INTERFACE I_JsonDeserializerChangedEvent EXTENDS I_Event

PROPERTY PUBLIC Target : I_JsonDeserializer
GET
END_GET
END_PROPERTY

END_INTERFACE

(* stored: Version 1.1.0.1, ProductVersion 3.1.4024.12
   Itf I_JsonDeserializerChangedEvent: Id {40baa505-43af-4f39-bb65-a6df1e3a04e2}
   Property Target: Id {c8ae607c-6e4e-4a76-b1e9-7059ebb604db}
   Get Get: Id {20fcb79e-8ff2-4317-a723-95b539d3c194} *)
